TEXTLIST TextList
   = ''
END_TEXTLIST

(* stored: Version 1.1.0.1, ProductVersion 3.1.4022.18
   TextList TextList: Id {466a9928-beed-4071-9dda-a74b267211d4} *)
